FUNCTION_BLOCK GET_AT_INDEX (* Fetch value from array at given index. Array data type has to match with output data type. *)
  (* Description: Copyright (c) 2014 Profactor GmbH This program and the accompanying materials are made available under the terms of the Eclipse Public License 2.0 which is available at https://www.eclipse.org/legal/epl-2.0/ SPDX-License-Identifier: EPL-2.0 *)
  (* Version 1.0, 2014-07-11, Matthias Plasch, Profactor GmbH *)
  (* Version 3.0, 2025-04-14, Patrick Aigner, changed package *)
  PACKAGE eclipse4diac::utils;
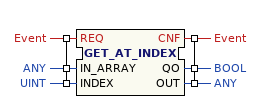
  EVENT_INPUT
    REQ WITH IN_ARRAY, INDEX; (* Service Request *)
  END_EVENT
  EVENT_OUTPUT
    CNF WITH QO, OUT; (* Confirmation of Requested Service *)
  END_EVENT
  VAR_INPUT
    IN_ARRAY : ANY; (* input array *)
    INDEX : UINT; (* index to fetch value from *)
  END_VAR
  VAR_OUTPUT
    QO : BOOL; (* Event Output Qualifier *)
    OUT : ANY; (* fetched output value *)
  END_VAR
END_FUNCTION_BLOCK
